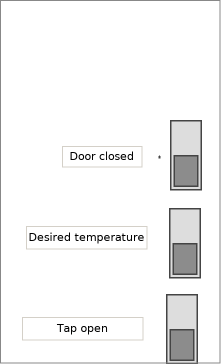
VISUALIZATION Visualization  // 221x364
    DipSwitch (151,156 17x1), behaviour: TOGGLE, style: Switch-DipSwitch-Gray
    DipSwitch (151,120 70x70), behaviour: TOGGLE, style: Switch-DipSwitch-Gray
    DipSwitch (150,208 70x70), behaviour: TOGGLE, style: Switch-DipSwitch-Gray
    DipSwitch (147,294 70x70), behaviour: TOGGLE, style: Switch-DipSwitch-Gray
    Textfield (62,146 80x21), "Door closed"
    Textfield (26,226 121x23), "Desired temperature"
    Textfield (22,317 121x23), "Tap open"
END_VISUALIZATION

(* stored: Version 1.1.0.1, ProductVersion 3.1.4024.12
   Visu Visualization: Id {00e66e05-e069-4c58-9ec9-a7d1fe57b791} *)
